# EPICS autosave request: iocBoot/ioc13bmd_pg1/auto_settings.req
file "spinnaker_settings.req",            P=$(P),  R=cam1:
file "NDStdArrays_settings.req",          P=$(P),  R=image1:
file "commonPlugin_settings.req",         P=$(P)
file "TomoCollect_settings.req",          P=$(P),  R=TC:
$(P)cam1:GC_OnBoaColProEna
$(P)cam1:GC_VideoMode
